{attribute 'GeneratedUsingTerminal: EP2028-0001-0016'}
{attribute addProperty BoxType "EP2028-0001-0016"}
{attribute addProperty Id "EtcSlaveTerminalBaseChannel_1AT %Q*Channel_42CA91F71Channel_2AT %Q*Channel_42CA91F71Channel_3AT %Q*Channel_42CA91F71Channel_4AT %Q*Channel_42CA91F71Channel_5AT %Q*Channel_42CA91F71Channel_6AT %Q*Channel_42CA91F71Channel_7AT %Q*Channel_42CA91F71Channel_8AT %Q*Channel_42CA91F71WcStateAT %I*WcState_0B2B16F91InfoDataAT %I*InfoData_6F19DB2B2"}
{attribute addProperty CRC "3630786787"}
{attribute addProperty Size "11"}
TYPE EP2028_D86968E3 EXTENDS EtcSlaveTerminalBase :
STRUCT
	{attribute addProperty Name "Channel_1"}
	Channel_1 : Channel_42CA91F7;
	{attribute addProperty Name "Channel_2"}
	Channel_2 : Channel_42CA91F7;
	{attribute addProperty Name "Channel_3"}
	Channel_3 : Channel_42CA91F7;
	{attribute addProperty Name "Channel_4"}
	Channel_4 : Channel_42CA91F7;
	{attribute addProperty Name "Channel_5"}
	Channel_5 : Channel_42CA91F7;
	{attribute addProperty Name "Channel_6"}
	Channel_6 : Channel_42CA91F7;
	{attribute addProperty Name "Channel_7"}
	Channel_7 : Channel_42CA91F7;
	{attribute addProperty Name "Channel_8"}
	Channel_8 : Channel_42CA91F7;
	{attribute addProperty Name "WcState"}
	WcState : WcState_0B2B16F9;
	{attribute addProperty Name "InfoData"}
	InfoData : InfoData_6F19DB2B;
END_STRUCT
END_TYPE

(* stored: Version 1.2.0.0, ProductVersion 3.1.4024.9
   DUT EP2028_D86968E3: Id {18ccca82-73e9-4a5b-a571-0cf0914267cf} *)
